FUNCTION_BLOCK FB_SlotList
VAR_INPUT
END_VAR
VAR_OUTPUT
END_VAR
VAR
	pHead	: POINTER TO ST_POINTER2;
	pTail	: POINTER TO ST_POINTER2;
	pCurrent: POINTER TO ST_POINTER2;
	nCount	: UINT;
END_VAR

PROPERTY P_nCount : UINT
GET
P_nCount := nCount;
END_GET
END_PROPERTY

METHOD M_GetAtIndex : POINTER TO FB_Slot
VAR_INPUT
	nIndex : UINT;
END_VAR

VAR
	i : UINT;
	pItem : POINTER TO ST_POINTER2;
END_VAR
//mit Index ist die fortlaufende Nummer eines Slots in der Liste gemeint
IF nIndex > 0 AND nIndex <= nCount THEN
	pItem := pHead;
	FOR i := 1 TO nIndex - 1 BY 1 DO
		pItem := pItem^.pNext;
	END_FOR
	M_GetAtIndex := pItem^.pContent;
END_IF
END_METHOD

METHOD M_GetAtNr : POINTER TO FB_Slot
VAR_INPUT
	nNr	: UINT;
END_VAR

VAR
	pPointer : POINTER TO ST_POINTER2;
	pSlot: POINTER TO FB_Slot; 
END_VAR
//Gibt Slot anhand der SlotNr zurück
pPointer := pHead;
WHILE pPointer > 0 DO
	pSlot := pPointer^.pContent;
	IF pSlot^.P_nNr = nNr THEN
		EXIT;
	ELSE
		pSlot := 0;
	END_IF
	pPointer := pPointer^.pNext;
END_WHILE

IF pSlot > 0 THEN
	M_GetAtNr := pSlot;
END_IF
END_METHOD

METHOD M_SetCurrentToHead : BOOL
VAR_INPUT
END_VAR
pCurrent := pHead;
END_METHOD

METHOD M_Add : ERRORID
VAR_INPUT
	pSlot : POINTER TO FB_Slot;
END_VAR

VAR
	pNew : POINTER TO ST_POINTER2;
END_VAR
pNew := pHead;
WHILE pNew > 0 DO
	IF pNew^.pContent = pSlot THEN
		M_Add := 43434;
		RETURN;
	END_IF
	pNew := pNew^.pNext;
END_WHILE

pNew := __NEW(ST_Pointer2);
MEMSET(pNew,0,SIZEOF(ST_POINTER2));
pNew^.pContent := pSlot;
IF pHead = 0 THEN
	pHead := pTail := pNew;
ELSE
	pNew^.pPrev := pTail; 
	pTail^.pNext := pNew;
	pTail := pNew;
END_IF
nCount := nCount + 1;
END_METHOD

METHOD M_Reset
VAR_INPUT
END_VAR

VAR
	pDelete : POINTER TO ST_Pointer2;
	pNext	: POINTER TO ST_Pointer2;
	pSlot	: POINTER TO FB_SLOT;
END_VAR
pDelete := pHead;
WHILE  pDelete > 0 DO
	pNext := pDelete^.pNext;
	pSlot := pDelete^.pContent; 
	IF pSlot > 0 THEN
		__DELETE(pSlot);
	END_IF
	__DELETE(pDelete);
	pDelete := pNext;
END_WHILE
pHead := 0;
pTail := 0;
pCurrent := 0;
nCount := 0;
END_METHOD

METHOD M_GetNext : POINTER TO FB_Slot
VAR_INPUT
END_VAR

VAR
	pSlot : POINTER TO FB_Slot;
END_VAR
IF pCurrent > 0 THEN
	pSlot := pCurrent^.pContent;
	IF pSlot > 0 THEN
		M_GetNext := pSlot;
	END_IF
	pCurrent := pCurrent^.pNext;
END_IF
END_METHOD

END_FUNCTION_BLOCK

(* stored: Version 1.1.0.1, ProductVersion 3.1.4020.12
   POU FB_SlotList: Id {4cf46d43-eef9-4d90-8049-5f264e9f812f}, SpecialFunc None
   Property P_nCount: Id {45fd7700-41a2-400a-bc4d-70474bee2ec5}
   Get Get: Id {1fc1a22f-8ddc-416f-8c98-dffec85b7854}
   Method M_GetAtIndex: Id {58b32ec9-e2fc-4380-a64f-5db5d0070ada}
   Method M_GetAtNr: Id {6f93f9bf-bedc-47fd-be1c-c7d58747dfde}
   Method M_SetCurrentToHead: Id {d23479f9-9c12-485a-a952-2fff5ea0c0d8}
   Method M_Add: Id {e21ecc7b-255a-4d0f-b14f-e8abb80fd21c}
   Method M_Reset: Id {f32da28c-fe0c-4c52-bf3d-875eab7ba948}
   Method M_GetNext: Id {f616f28b-5554-4d7c-9265-cae37f0f0333} *)
